TYPE ST_CommandChangeMode :
STRUCT
	cmdChangeProduction	 	  	: FB_CommandChangeProduction;
	cmdChangeMaintenance		: FB_CommandChangeMaintenance;
	cmdChangeManual		    	: FB_CommandChangeManual;
	cmdChangeWashing		   	: FB_CommandChangeWashing;
	cmdChangeDiagnostics		: FB_CommandChangeDiagnostics;
END_STRUCT
END_TYPE

(* stored: Version 1.1.0.1
   DUT ST_CommandChangeMode: Id {b75752ec-7f06-0c94-055d-596f76bcbf81} *)
